// TIA Portal V18 export
DATA_BLOCK "IEC_Counter_0_DB"   // DB11
{ S7_Optimized_Access := 'TRUE' }
// stored: AutoNumber true, InstanceOfName IEC_UCOUNTER, OfSystemLibElement IEC_UCOUNTER, OfSystemLibVersion 1.0
"IEC_UCOUNTER"
   // VAR RETAIN
   //    CU : Bool;
   //    CD : Bool;
   //    R : Bool;
   //    LD : Bool;
   //    QU : Bool;
   //    QD : Bool;
   //    PV : UInt;
   //    CV : UInt;
   // END_VAR
BEGIN
END_DATA_BLOCK
